// TIA Portal project "2022.06.07_移动指令的用法" (V17)

(* hardware
DEVICE "S7-1200 station_1"  S7-1200 Station
   slot 0: "Rack_0"  S7-1200 Rack  Rack  V1.0
   slot 1: "PLC_1"  CPU 1212C DC/DC/DC  6ES7 212-1AE40-0XB0  V4.5
*)

// ===== PLC "PLC_1"  CPU 1212C DC/DC/DC =====

VAR_GLOBAL   // PLC tag table "默认变量表"
   "模拟量输入" AT %MW100 : Word;
   "Tag_3" AT %MW102 : UInt;
   "Tag_4" AT %MW104 : UInt;
   "Tag_5" AT %MW106 : UInt;
   "Tag_6" AT %I0.0 : Bool;
   "Tag_7" AT %M0.0 : Bool;
   "X(2)" AT %MW10 : Word;
   "Tag_9" AT %MW12 : UInt;
   "X" AT %MW0 : Word;
   "a" AT %MW2 : Word;
   "b" AT %MW4 : Int;
   "c" AT %MW8 : Int;
   "实时温度" AT %MD0 : Real;
   "Tag_10" AT %MD2 : Real;
   "f" AT %MD4 : Real;
   "g" AT %MD8 : Real;
   "X(1)" AT %MD12 : Real;
   "Tag_8" AT %MD16 : Real;
   "中间值(1)" AT %MD200 : Real;
   "中间值" AT %MD104 : Real;
   "工程值" AT %MD108 : Real;
   "要求的频率" AT %MD60 : Real;
   "百分比" AT %MD64 : Real;
   "Tag_12" AT %MW70 : Int;
   "Tag_2" AT %I0.1 : Bool;
   "0" AT %Q0.0 : Bool;
   "加热" AT %Q0.1 : Bool;
   "Tag_1" AT %MD100 : Time;
   "Tag_11" AT %M0.1 : Bool;
   "Tag_13" AT %QB0 : Byte;
END_VAR

DATA_BLOCK "测试数据块_1"   // DB1
{ S7_Optimized_Access := 'FALSE' }
VERSION : 0.1
BEGIN
END_DATA_BLOCK

// folder: System blocks/Program resources

DATA_BLOCK "IEC_Timer_0_DB"   // DB2
{ S7_Optimized_Access := 'TRUE' }
AUTHOR : Simatic
FAMILY : IEC
NAME : IEC_TMR
VERSION : 1.0
// stored: InstanceOfName IEC_TIMER
"IEC_TIMER"
BEGIN
END_DATA_BLOCK

// folder: (top level)

ORGANIZATION_BLOCK "Main"   // OB1, LAD, ProgramCycle
TITLE = "Main Program Sweep (Cycle)"
{ S7_Optimized_Access := 'TRUE' }
VERSION : 0.1
   VAR_INPUT
      Initial_Call : Bool;   // Initial call of this OB
      Remanence : Bool;   // =True, if remanent data are available
   END_VAR
BEGIN

REGION Network 1
   // 启动：q0.0-0.2-0.4-0.6亮，1秒后，1.3.5.7亮，3s后全亮
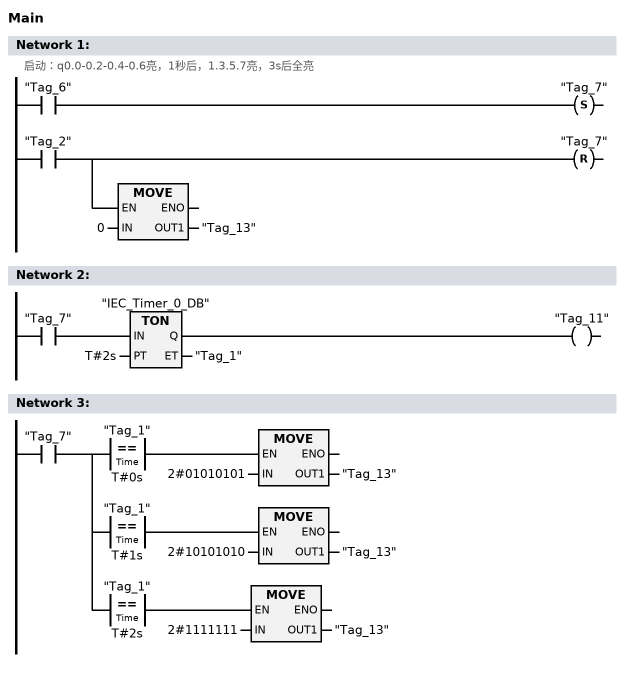
   RUNG wire#powerrail
      Contact( "Tag_6" )
      S_Coil( "Tag_7" )
   END_RUNG
   RUNG wire#powerrail
      Contact( "Tag_2" )
      wire#w1
      R_Coil( "Tag_7" )
   END_RUNG
   RUNG wire#w1
      Move(in := 0, out1 => "Tag_13")
   END_RUNG
   // the same network as SCL:
   IF "Tag_6" THEN "Tag_7" := TRUE; END_IF;
   IF "Tag_2" THEN
       "Tag_7" := FALSE;
       "Tag_13" := 0;
   END_IF;
END_REGION

REGION Network 2
   "IEC_Timer_0_DB".TON(IN := "Tag_7", PT := T#2s, ET => "Tag_1");
   "Tag_11" := "IEC_Timer_0_DB".Q;
END_REGION

REGION Network 3
   RUNG wire#powerrail
      Contact( "Tag_7" )
      wire#w1
      { S7_Templates := "SrcType := Time" } EQ_Contact(in1 := "Tag_1", in2 := T#0s)
      Move(in := 2#01010101, out1 => "Tag_13")
   END_RUNG
   RUNG wire#w1
      { S7_Templates := "SrcType := Time" } EQ_Contact(in1 := "Tag_1", in2 := T#1s)
      Move(in := 2#10101010, out1 => "Tag_13")
   END_RUNG
   RUNG wire#w1
      { S7_Templates := "SrcType := Time" } EQ_Contact(in1 := "Tag_1", in2 := T#2s)
      Move(in := 2#1111111, out1 => "Tag_13")
   END_RUNG
   // the same network as SCL:
   IF "Tag_7" AND ("Tag_1" = T#0s) THEN "Tag_13" := 2#01010101; END_IF;
   IF "Tag_7" AND ("Tag_1" = T#1s) THEN "Tag_13" := 2#10101010; END_IF;
   IF "Tag_7" AND ("Tag_1" = T#2s) THEN "Tag_13" := 2#1111111; END_IF;
END_REGION
END_ORGANIZATION_BLOCK